// Interlock logic for the Amphos attenuator
FUNCTION F_AmphosAttenuatorEnable : BOOL
VAR_INPUT
    bAmphosOn : BOOL; // Whether the Amphos is turned on
END_VAR
VAR_IN_OUT CONSTANT
    stErrors : ST_ErrorStates; // Currently detected errors
END_VAR
VAR
END_VAR

IF stErrors.bHardwareFailure // Close attenuator if there is a hardware failure
    OR NOT bAmphosOn // Close attenuator if Amphos is not on
    OR stErrors.bLeakOpticalTableAmphosOn OR stErrors.bLeakOpcpaCarbideOn OR stErrors.bLeakUnderTable // Close attenuator if there is a leak on the optical table with amphos on, there is a leak in the OPCPA with the carbide on, or there is a leak under the table
    (* OR stErrors.bAmphosMRC01 // Close attenuator if there is an AmphosMRC01 error *)
THEN
    F_AmphosAttenuatorEnable := FALSE;
ELSE
    F_AmphosAttenuatorEnable := TRUE;
END_IF

END_FUNCTION

(* stored: Version 1.1.0.1, ProductVersion 3.1.4022.18
   POU F_AmphosAttenuatorEnable: Id {7ab6d45d-4336-488b-ae1d-ec9e617ae7af}, SpecialFunc None *)
